PROGRAM F21_ContentHandScanner_ORG
VAR
	fbBarcodeType			: FB_SYSTEM_BarcodeType;

	bPackBarcode					: BOOL;
	bOuterIntermediateBarcode		: BOOL;
	bOuterBarcode					: BOOL;
	bCaseBarcode					: BOOL;
	sPackBarcode					: T_PACK_Barcode;
	sOuterIntermediateBarcode		:  T_MaxString;
	sOuterBarcode					: T_OUTER_Barcode;
	sCaseBarcode					: T_CASE_Barcode;

	fbSearchCaseContent	: FB_SYSTEM_SearchBarcode;

	fbFindOACFile			: FB_OAC_FindFile;
	fbFindOCVFile			: FB_OCV_FindFile;
	stOACData				: ST_OAC_Data;
	strCode				: T_PACK_Barcode;
	strOACFile				: T_OAC_Filename;
	strOCVFile				: T_OCV_Filename;


	fbMoveCACFromArchive	: FB_CAC_MoveFromArchive;

	strCACFile				: T_CAC_Filename;

	bOACFound: BOOL;
	bOCVFound: BOOL;
	bOCVValid: BOOL;
	strOuterCodeAI:			STRING(255);
	(*strPackCodeAI:			STRING(255);*)

	bValidateForOCVDataExistDone :BOOL;
	bValidateForRefeedDone: BOOL;
	bValidateForRefeedOK: BOOL;

	rtrigValidateOCVForDataExistValid			: R_TRIG;
	rtrigValidateOCVForDataExistInvalid			: R_TRIG;
	rtrigValidateOCVForDataNotExist			: R_TRIG;
	tofValidateOCVForDataExisValid			: TOF;
	tofValidateOCVForDataExisInvalid			: TOF;
	tofValidateOCVForDataNotExis				: TOF;


	rtrigValidateOACForRefeedDoneValid		: R_TRIG;
	rtrigValidateOACForRefeedDoneInvalid		: R_TRIG;
	rtrigValidateOACForDataNotExist			: R_TRIG;
	tofValidateOACForRefeedValid			: TOF;
	tofValidateOACForRefeedInvalid			: TOF;
	tofValidateOACForDataNotExis				: TOF;

	rtrigRestoreCACFileDoneValid: R_TRIG;
	rtrigRestoreCACFileDoneInvalid: R_TRIG;
	tofRestoreCACFileValid: TOF;
	tofRestoreCACFileInvalid: TOF;

END_VAR

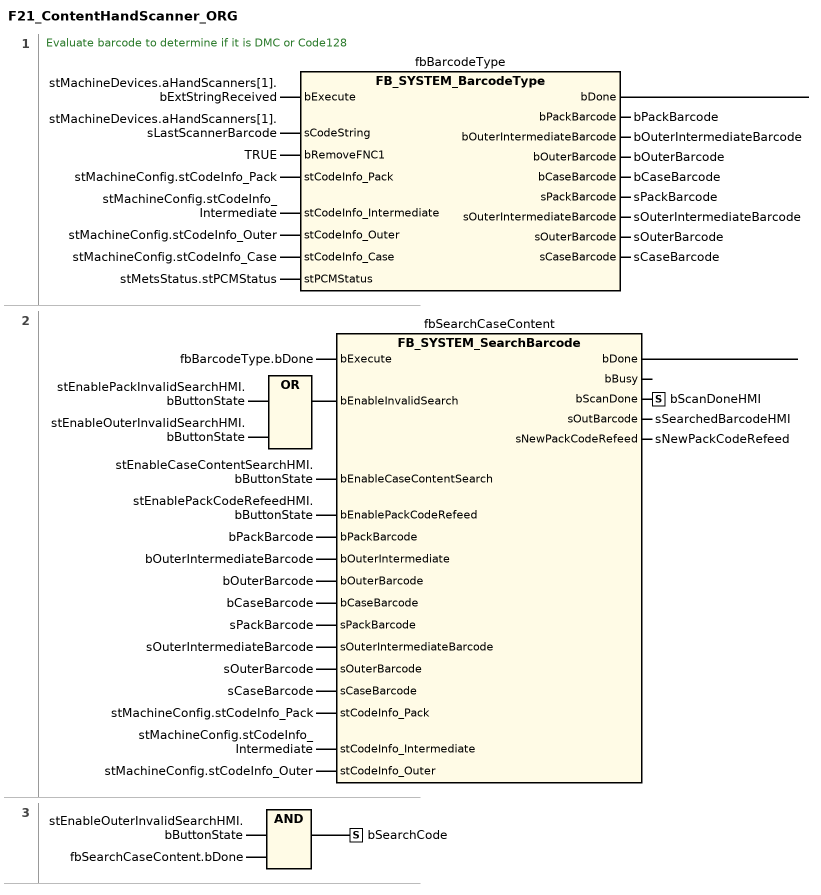
// NETWORK 1
// Evaluate barcode to determine if it is DMC or Code128
fbBarcodeType(
    bExecute := stMachineDevices.aHandScanners[1].bExtStringReceived,
    sCodeString := stMachineDevices.aHandScanners[1].sLastScannerBarcode,
    bRemoveFNC1 := TRUE,
    stCodeInfo_Pack := stMachineConfig.stCodeInfo_Pack,
    stCodeInfo_Intermediate := stMachineConfig.stCodeInfo_Intermediate,
    stCodeInfo_Outer := stMachineConfig.stCodeInfo_Outer,
    stCodeInfo_Case := stMachineConfig.stCodeInfo_Case,
    stPCMStatus := stMetsStatus.stPCMStatus,
    bPackBarcode => bPackBarcode,
    bOuterIntermediateBarcode => bOuterIntermediateBarcode,
    bOuterBarcode => bOuterBarcode,
    bCaseBarcode => bCaseBarcode,
    sPackBarcode => sPackBarcode,
    sOuterIntermediateBarcode => sOuterIntermediateBarcode,
    sOuterBarcode => sOuterBarcode,
    sCaseBarcode => sCaseBarcode); // FB_SYSTEM_BarcodeType

// NETWORK 2
fbSearchCaseContent(
    bExecute := fbBarcodeType.bDone,
    bEnableInvalidSearch := stEnablePackInvalidSearchHMI.bButtonState OR stEnableOuterInvalidSearchHMI.bButtonState,
    bEnableCaseContentSearch := stEnableCaseContentSearchHMI.bButtonState,
    bEnablePackCodeRefeed := stEnablePackCodeRefeedHMI.bButtonState,
    bPackBarcode := bPackBarcode,
    bOuterIntermediate := bOuterIntermediateBarcode,
    bOuterBarcode := bOuterBarcode,
    bCaseBarcode := bCaseBarcode,
    sPackBarcode := sPackBarcode,
    sOuterIntermediateBarcode := sOuterIntermediateBarcode,
    sOuterBarcode := sOuterBarcode,
    sCaseBarcode := sCaseBarcode,
    stCodeInfo_Pack := stMachineConfig.stCodeInfo_Pack,
    stCodeInfo_Intermediate := stMachineConfig.stCodeInfo_Intermediate,
    stCodeInfo_Outer := stMachineConfig.stCodeInfo_Outer,
    sOutBarcode => sSearchedBarcodeHMI,
    sNewPackCodeRefeed => sNewPackCodeRefeed); // FB_SYSTEM_SearchBarcode
bScanDoneHMI S= fbSearchCaseContent.bScanDone;

// NETWORK 3
bSearchCode S= stEnableOuterInvalidSearchHMI.bButtonState AND fbSearchCaseContent.bDone;

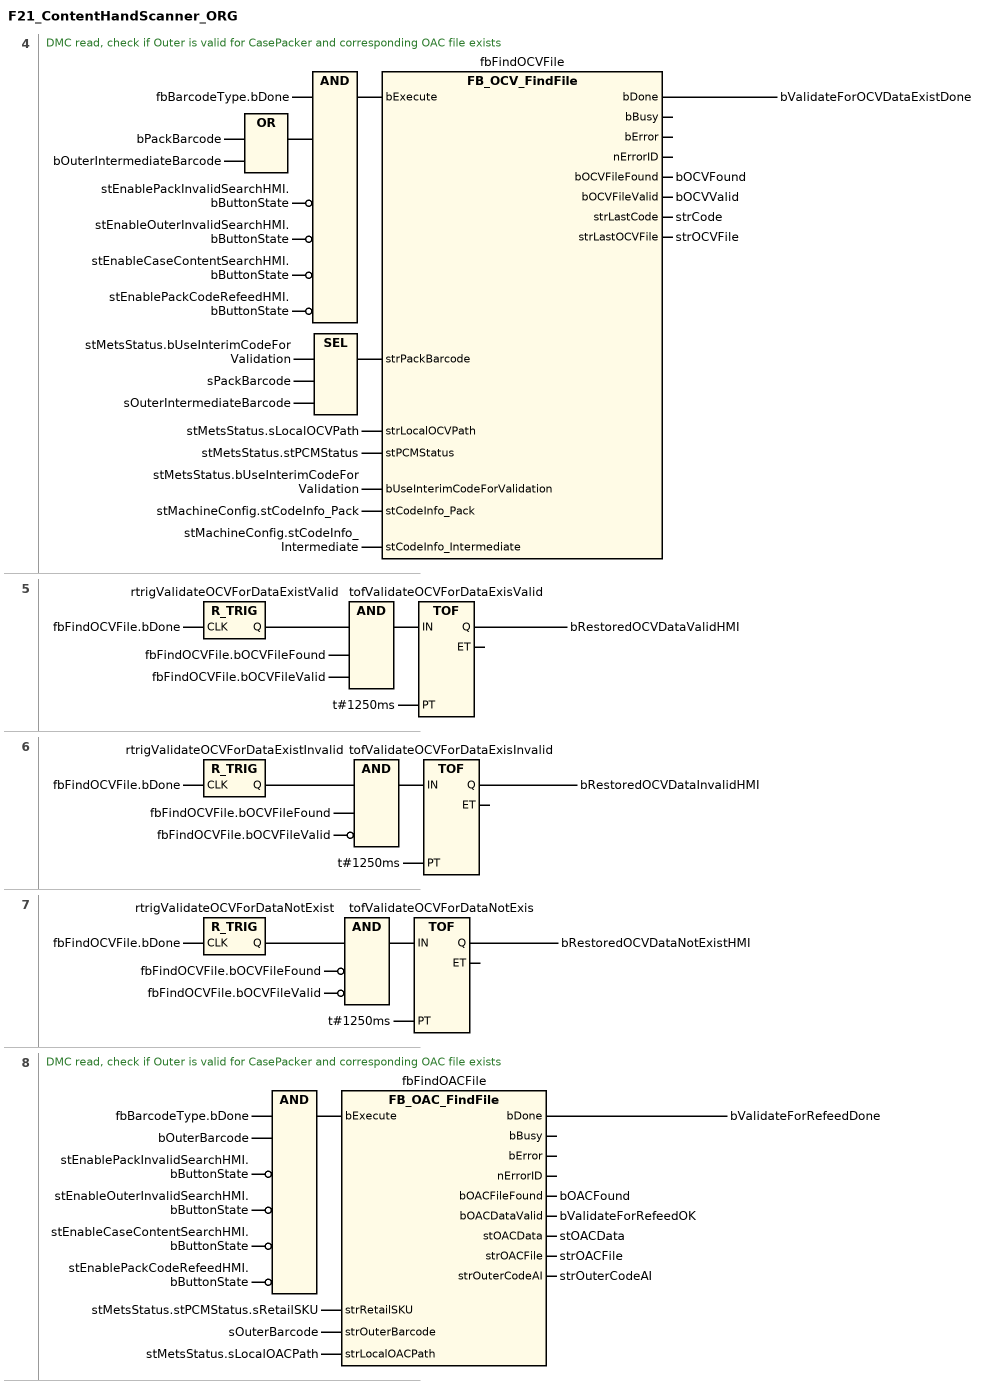
// NETWORK 4
// DMC read, check if Outer is valid for CasePacker and corresponding OAC file exists
fbFindOCVFile(
    bExecute := fbBarcodeType.bDone AND (bPackBarcode OR bOuterIntermediateBarcode) AND NOT stEnablePackInvalidSearchHMI.bButtonState AND NOT stEnableOuterInvalidSearchHMI.bButtonState AND NOT stEnableCaseContentSearchHMI.bButtonState AND NOT stEnablePackCodeRefeedHMI.bButtonState,
    strPackBarcode := SEL(stMetsStatus.bUseInterimCodeForValidation, sPackBarcode, sOuterIntermediateBarcode),
    strLocalOCVPath := stMetsStatus.sLocalOCVPath,
    stPCMStatus := stMetsStatus.stPCMStatus,
    bUseInterimCodeForValidation := stMetsStatus.bUseInterimCodeForValidation,
    stCodeInfo_Pack := stMachineConfig.stCodeInfo_Pack,
    stCodeInfo_Intermediate := stMachineConfig.stCodeInfo_Intermediate,
    bOCVFileFound => bOCVFound,
    bOCVFileValid => bOCVValid,
    strLastCode => strCode,
    strLastOCVFile => strOCVFile); // FB_OCV_FindFile
bValidateForOCVDataExistDone := fbFindOCVFile.bDone;

// NETWORK 5
rtrigValidateOCVForDataExistValid(CLK := fbFindOCVFile.bDone); // R_TRIG
tofValidateOCVForDataExisValid(IN := rtrigValidateOCVForDataExistValid.Q AND fbFindOCVFile.bOCVFileFound AND fbFindOCVFile.bOCVFileValid, PT := t#1250ms); // TOF
bRestoredOCVDataValidHMI := tofValidateOCVForDataExisValid.Q;

// NETWORK 6
rtrigValidateOCVForDataExistInvalid(CLK := fbFindOCVFile.bDone); // R_TRIG
tofValidateOCVForDataExisInvalid(IN := rtrigValidateOCVForDataExistInvalid.Q AND fbFindOCVFile.bOCVFileFound AND NOT fbFindOCVFile.bOCVFileValid, PT := t#1250ms); // TOF
bRestoredOCVDataInvalidHMI := tofValidateOCVForDataExisInvalid.Q;

// NETWORK 7
rtrigValidateOCVForDataNotExist(CLK := fbFindOCVFile.bDone); // R_TRIG
tofValidateOCVForDataNotExis(IN := rtrigValidateOCVForDataNotExist.Q AND NOT fbFindOCVFile.bOCVFileFound AND NOT fbFindOCVFile.bOCVFileValid, PT := t#1250ms); // TOF
bRestoredOCVDataNotExistHMI := tofValidateOCVForDataNotExis.Q;

// NETWORK 8
// DMC read, check if Outer is valid for CasePacker and corresponding OAC file exists
fbFindOACFile(
    bExecute := fbBarcodeType.bDone AND bOuterBarcode AND NOT stEnablePackInvalidSearchHMI.bButtonState AND NOT stEnableOuterInvalidSearchHMI.bButtonState AND NOT stEnableCaseContentSearchHMI.bButtonState AND NOT stEnablePackCodeRefeedHMI.bButtonState,
    strRetailSKU := stMetsStatus.stPCMStatus.sRetailSKU,
    strOuterBarcode := sOuterBarcode,
    strLocalOACPath := stMetsStatus.sLocalOACPath,
    bOACFileFound => bOACFound,
    bOACDataValid => bValidateForRefeedOK,
    stOACData => stOACData,
    strOACFile => strOACFile,
    strOuterCodeAI => strOuterCodeAI); // FB_OAC_FindFile
bValidateForRefeedDone := fbFindOACFile.bDone;

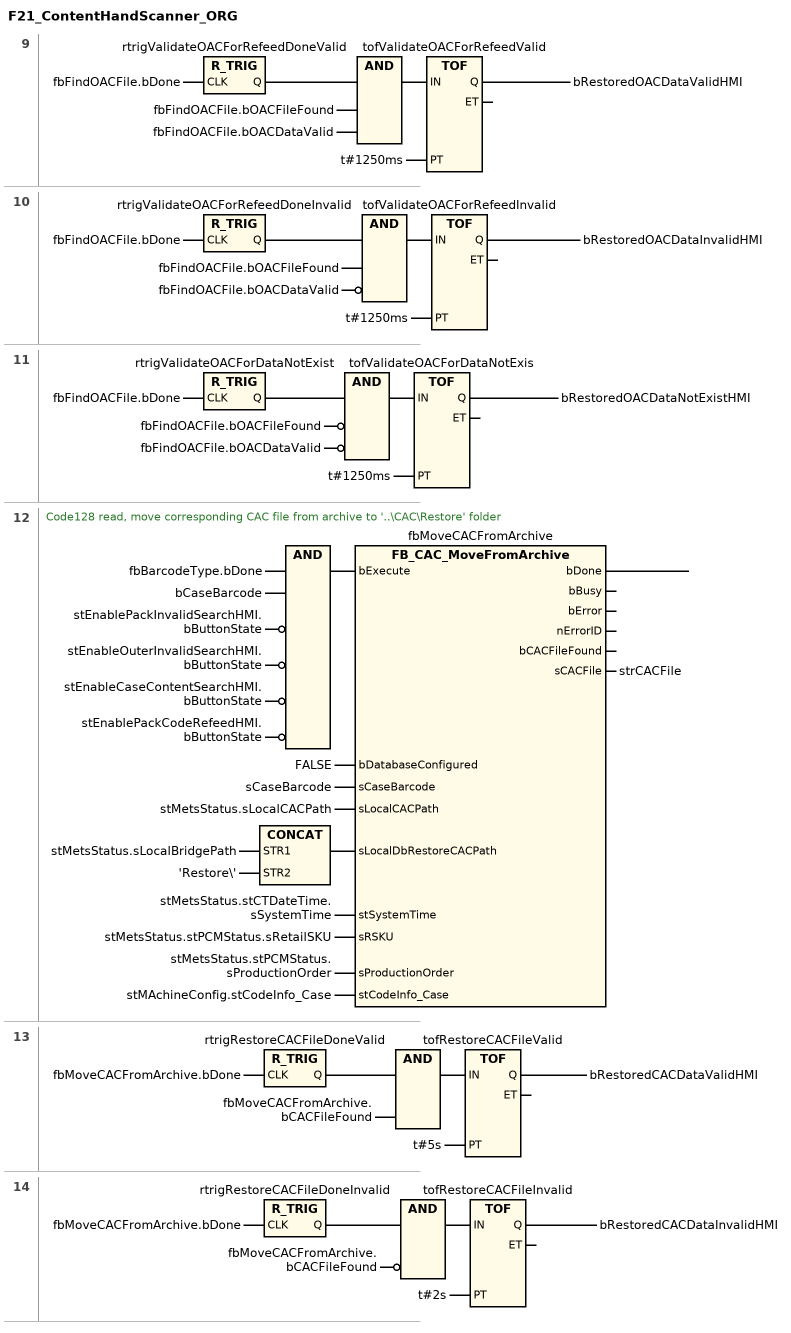
// NETWORK 9
rtrigValidateOACForRefeedDoneValid(CLK := fbFindOACFile.bDone); // R_TRIG
tofValidateOACForRefeedValid(IN := rtrigValidateOACForRefeedDoneValid.Q AND fbFindOACFile.bOACFileFound AND fbFindOACFile.bOACDataValid, PT := t#1250ms); // TOF
bRestoredOACDataValidHMI := tofValidateOACForRefeedValid.Q;

// NETWORK 10
rtrigValidateOACForRefeedDoneInvalid(CLK := fbFindOACFile.bDone); // R_TRIG
tofValidateOACForRefeedInvalid(IN := rtrigValidateOACForRefeedDoneInvalid.Q AND fbFindOACFile.bOACFileFound AND NOT fbFindOACFile.bOACDataValid, PT := t#1250ms); // TOF
bRestoredOACDataInvalidHMI := tofValidateOACForRefeedInvalid.Q;

// NETWORK 11
rtrigValidateOACForDataNotExist(CLK := fbFindOACFile.bDone); // R_TRIG
tofValidateOACForDataNotExis(IN := rtrigValidateOACForDataNotExist.Q AND NOT fbFindOACFile.bOACFileFound AND NOT fbFindOACFile.bOACDataValid, PT := t#1250ms); // TOF
bRestoredOACDataNotExistHMI := tofValidateOACForDataNotExis.Q;

// NETWORK 12
// Code128 read, move corresponding CAC file from archive to '..\CAC\Restore' folder
fbMoveCACFromArchive(
    bExecute := fbBarcodeType.bDone AND bCaseBarcode AND NOT stEnablePackInvalidSearchHMI.bButtonState AND NOT stEnableOuterInvalidSearchHMI.bButtonState AND NOT stEnableCaseContentSearchHMI.bButtonState AND NOT stEnablePackCodeRefeedHMI.bButtonState,
    bDatabaseConfigured := FALSE,
    sCaseBarcode := sCaseBarcode,
    sLocalCACPath := stMetsStatus.sLocalCACPath,
    sLocalDbRestoreCACPath := CONCAT(STR1 := stMetsStatus.sLocalBridgePath, STR2 := 'Restore\'),
    stSystemTime := stMetsStatus.stCTDateTime.sSystemTime,
    sRSKU := stMetsStatus.stPCMStatus.sRetailSKU,
    sProductionOrder := stMetsStatus.stPCMStatus.sProductionOrder,
    stCodeInfo_Case := stMAchineConfig.stCodeInfo_Case,
    sCACFile => strCACFile); // FB_CAC_MoveFromArchive

// NETWORK 13
rtrigRestoreCACFileDoneValid(CLK := fbMoveCACFromArchive.bDone); // R_TRIG
tofRestoreCACFileValid(IN := rtrigRestoreCACFileDoneValid.Q AND fbMoveCACFromArchive.bCACFileFound, PT := t#5s); // TOF
bRestoredCACDataValidHMI := tofRestoreCACFileValid.Q;

// NETWORK 14
rtrigRestoreCACFileDoneInvalid(CLK := fbMoveCACFromArchive.bDone); // R_TRIG
tofRestoreCACFileInvalid(IN := rtrigRestoreCACFileDoneInvalid.Q AND NOT fbMoveCACFromArchive.bCACFileFound, PT := t#2s); // TOF
bRestoredCACDataInvalidHMI := tofRestoreCACFileInvalid.Q;

END_PROGRAM

(* stored: Version 1.1.0.1, ProductVersion 3.1.4024.15
   POU F21_ContentHandScanner_ORG: Id {1d9a71e0-5404-4e96-8df2-ca02f4244ac3}, SpecialFunc None *)
